INTERFACE IPointerComparer EXTENDS IObject

METHOD Compare : COMPARISION_RESULT
VAR_INPUT
	left : PVOID;
	right : PVOID;
END_VAR
END_METHOD

END_INTERFACE

(* stored: Version 1.1.0.1
   Itf IPointerComparer: Id {26f7205f-8930-4fff-99d1-ce7c2b42125c}
   Method Compare: Id {b70a82e2-80c6-403b-a1e0-841574c87ebf} *)
